{attribute addProperty BoxType "EP2816-0004-0016"}
{attribute addProperty Id "DO_Outputs_ChannelAT %Q*ARRAY[0..8] OF DO_Outputs_Channel_33B76376128160WcStateAT %I*WcState_28A8677510.1250InfoDataAT %I*InfoData_BC63D37F80100"}
{attribute addProperty CRC "1412542612"}
{attribute addProperty SizeInBites "209"}
{attribute addProperty SizeInBytes "26.125"}
TYPE EP2816_68098FB0 :
STRUCT
	{attribute addProperty Name "DO_Outputs_Channel"}
	DO_Outputs_Channel : ARRAY[0..8] OF DO_Outputs_Channel_33B76376;
	{attribute addProperty Name "WcState"}
	WcState : WcState_28A86775;
	{attribute addProperty Name "InfoData"}
	InfoData : InfoData_BC63D37F;
END_STRUCT
END_TYPE

(* stored: Version 1.2.0.0, ProductVersion 3.1.4024.9
   DUT EP2816_68098FB0: Id {1384cec0-6b4b-4ab3-a603-2f3ccf4e8a05} *)
